% RSLogix 500 project MICROLOGIX 1000 CONVEYER MERGE_BAK002.RSS, saved by version 11.00.00.00 %
PROJECT "1000"    % processor: MicroLogix 1000 %

PROGRAM FILES
  LAD 2 "MAIN_PROG"  8 rungs
  LAD 3 "USER_FAULT"  1 rungs
  LAD 4 "HSC_INT"  1 rungs
  LAD 5 "STI_INT"  1 rungs
  LAD 6, 7, 8, 9, 10, 11, 12, 13, 14, 15, 16: only END

DATA FILES
  O0 OUTPUT  1 elements
  I1 INPUT  2 elements
  S2 STATUS  33 elements
  B3 BINARY  32 elements
  T4 TIMER  40 elements
  C5 COUNTER  32 elements
  R6 CONTROL  16 elements
  N7 INTEGER  105 elements

LADDER 2 "MAIN_PROG"
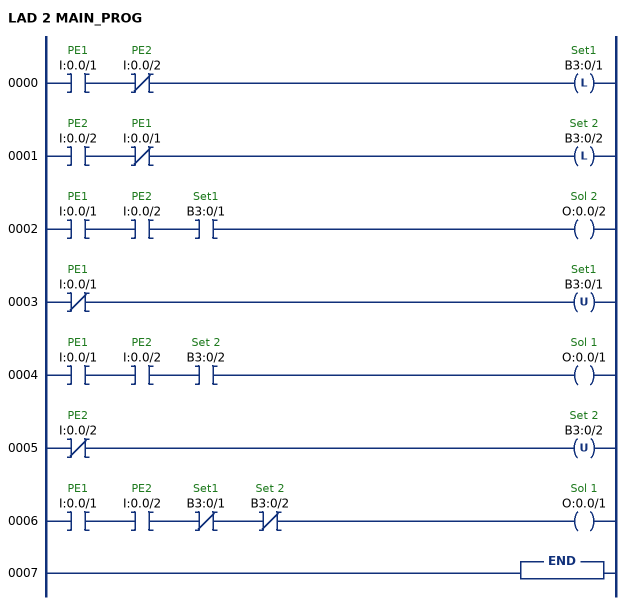
% Rung: 0 %
SOR XIC I:0.0/1 XIO I:0.0/2 OTL B3:0/1 EOR
%   I:0.0/1  "PE1" %
%   I:0.0/2  "PE2" %
%   B3:0/1  "Set1" %
% Rung: 1 %
SOR XIC I:0.0/2 XIO I:0.0/1 OTL B3:0/2 EOR
%   I:0.0/2  "PE2" %
%   I:0.0/1  "PE1" %
%   B3:0/2  "Set 2" %
% Rung: 2 %
SOR XIC I:0.0/1 XIC I:0.0/2 XIC B3:0/1 OTE O:0.0/2 EOR
%   I:0.0/1  "PE1" %
%   I:0.0/2  "PE2" %
%   B3:0/1  "Set1" %
%   O:0.0/2  "Sol 2" %
% Rung: 3 %
SOR XIO I:0.0/1 OTU B3:0/1 EOR
%   I:0.0/1  "PE1" %
%   B3:0/1  "Set1" %
% Rung: 4 %
SOR XIC I:0.0/1 XIC I:0.0/2 XIC B3:0/2 OTE O:0.0/1 EOR
%   I:0.0/1  "PE1" %
%   I:0.0/2  "PE2" %
%   B3:0/2  "Set 2" %
%   O:0.0/1  "Sol 1" %
% Rung: 5 %
SOR XIO I:0.0/2 OTU B3:0/2 EOR
%   I:0.0/2  "PE2" %
%   B3:0/2  "Set 2" %
% Rung: 6 %
SOR XIC I:0.0/1 XIC I:0.0/2 XIO B3:0/1 XIO B3:0/2 OTE O:0.0/1 EOR
%   I:0.0/1  "PE1" %
%   I:0.0/2  "PE2" %
%   B3:0/1  "Set1" %
%   B3:0/2  "Set 2" %
%   O:0.0/1  "Sol 1" %
% Rung: 7 %
SOR END EOR

OTHER DOCUMENTED ADDRESSES
  B3:0/3  "Set 3"
